PROGRAM MAIN
VAR
END_VAR

Manual();
Auto();
TextDisplay();

END_PROGRAM

(* stored: Version 1.1.0.1, ProductVersion 3.1.4024.12
   POU MAIN: Id {db0c931c-047a-4f4f-8f5e-88ee12d2dd6d}, SpecialFunc None *)
